FUNCTION_BLOCK Test_F_Equals EXTENDS T_UnitTestBase
VAR
	Assertion : T_Assertion;
END_VAR

{attribute 'analysis' := '-33'} // inhibit unused variable warning
METHOD RunTest
VAR_OUTPUT
    TestCompleted : BOOL;
    TestFailed    : BOOL;
END_VAR
TestFailed S= NOT Assertion.AssertEquals_BOOL(Source    := TestName,
                             Expected := TRUE,
                            Actual   := F_Equals(1.000_005,
                                                 1.000_004,
                                                 0.000_002),
                            VariableName := 'F_Equals');

TestFailed S= NOT Assertion.AssertEquals_BOOL(Source    := TestName,
                             Expected := FALSE,
                            Actual   := F_Equals(1.000_005,
                                                 1.000_003,
                                                 0.000_001),
                            VariableName := 'F_Equals');

TestCompleted := TRUE;
END_METHOD

END_FUNCTION_BLOCK

(* stored: Version 1.1.0.1, ProductVersion 3.1.4024.12
   POU Test_F_Equals: Id {d450eb35-6669-43c3-b7d1-9542fcdbe9ff}, SpecialFunc None
   Method RunTest: Id {d92ffd0c-5320-4118-9797-c20d6d917275} *)
